	bDone									:BOOL;
	bBusy									:BOOL;
	bErr									:BOOL;
	nErrID									:UDINT;
	
END_VAR
VAR_IN_OUT

	stAxis									:Tc2_MC2.Axis_Ref;

END_VAR
VAR
	
	eStateRevSeq							:E_AxisReversingSequence;
	eRevSeqErrStep							:E_AxisReversingSequence := eAxisRevSeq_NoError;
	fbTimerIdleTime							:TON;
	fbMoveAbsolute							:Tc2_MC2.MC_MoveAbsolute;
	fbStop									:Tc2_MC2.MC_Stop;

END_VAR
(* End *)

(* Reversing sequence axis *)

	CASE eStateRevSeq OF

		eAxisRevSeq_Start			:	(* Wait for start *)
		
			bDone := FALSE;
			bBusy := FALSE;
			
			IF bStart
			THEN

				bBusy 		 := TRUE;
				eStateRevSeq := eAxisRevSeq_Init;
				
			END_IF		


		eAxisRevSeq_Init			:	(* Initialize *)
		
			fbMoveAbsolute(
				Axis	 := stAxis, 
				Execute	 := FALSE);
				
			fbTimerIdleTime(
				IN	 	 :=	FALSE);
			
			fbStop(
				Axis	 :=	stAxis,
				Execute	 :=	FALSE);
				
			eStateRevSeq := eAxisRevSeq_AxisStartPos1;


		eAxisRevSeq_AxisStartPos1	:	(* Start axis to position 1 *)
		
			fbMoveAbsolute(
				Axis		:= stAxis, 
				Execute		:= TRUE, 
				Position	:= fTargetPosition1, 
				Velocity	:= fTargetVelocity1, 
				ErrorID		=> nErrID);
			
		
			IF NOT fbMoveAbsolute.Busy
				AND NOT fbMoveAbsolute.Error
			THEN
			
				fbMoveAbsolute(
					Axis		:= stAxis, 
					Execute		:= FALSE);
				eStateRevSeq := eAxisRevSeq_IdleTime1;

			ELSIF bStop
			THEN

				fbMoveAbsolute(
					Axis	 := stAxis, 
					Execute	 := FALSE);
				eStateRevSeq := eAxisRevSeq_AxisStop;

			ELSIF NOT fbMoveAbsolute.Busy
					AND fbMoveAbsolute.Error
			THEN

				eRevSeqErrStep := eStateRevSeq;
				eStateRevSeq   := eAxisRevSeq_ErrorStep;

			END_IF


		eAxisRevSeq_IdleTime1		:	(* delayed restart *)
		
			fbTimerIdleTime(
				IN	:=	TRUE, 
				PT	:= 	tIdleTime);

			IF NOT bStop			
				AND fbTimerIdleTime.Q 
			THEN

				fbTimerIdleTime(IN	:=	FALSE);
				eStateRevSeq := eAxisRevSeq_AxisStartPos2;

			ELSIF bStop
			THEN

				eStateRevSeq := eAxisRevSeq_Done;

			END_IF


		eAxisRevSeq_AxisStartPos2	:	(* Start axis to position 2 *)
		
			fbMoveAbsolute(
				Axis		:= stAxis, 
				Execute		:= TRUE, 
				Position	:= fTargetPosition2, 
				Velocity	:= fTargetVelocity2, 
				ErrorID		=> nErrID);
			
		
			IF NOT fbMoveAbsolute.Busy
				AND NOT fbMoveAbsolute.Error
			THEN
				fbMoveAbsolute(
					Axis	 := stAxis, 
					Execute	 := FALSE);
				eStateRevSeq := eAxisRevSeq_IdleTime2;

			ELSIF bStop
			THEN

				fbMoveAbsolute(
					Axis		:= stAxis, 
					Execute	:= FALSE);
				eStateRevSeq := eAxisRevSeq_AxisStop;

			ELSIF NOT fbMoveAbsolute.Busy
					AND fbMoveAbsolute.Error
			THEN

				eRevSeqErrStep := eStateRevSeq;
				eStateRevSeq   := eAxisRevSeq_ErrorStep;

			END_IF		


		eAxisRevSeq_IdleTime2		:	(* delayed restart*)

			fbTimerIdleTime(
				IN	:=	TRUE, 
				PT	:= 	tIdleTime);
				
			IF NOT bStop			
				AND fbTimerIdleTime.Q 
			THEN

				fbTimerIdleTime(IN	:=	FALSE);
				eStateRevSeq := eAxisRevSeq_Done;
				
			ELSIF bStop
			THEN
			
				eStateRevSeq := eAxisRevSeq_Done;
				
			END_IF
			
			
		eAxisRevSeq_AxisStop		:	(* Stop axis *)

			fbStop(
				Axis	:=	stAxis, 
				Execute	:=	TRUE, 
				ErrorID	=>	nErrID );
				
			IF (fbStop.Done
				OR fbStop.CommandAborted)
				AND NOT fbStop.Error
			THEN
				fbStop(
					Axis	:=	stAxis, 
					Execute	:=	FALSE);
				eStateRevSeq := eAxisRevSeq_Done;

			ELSIF NOT fbStop.Busy
					AND fbStop.Error
			THEN

				eRevSeqErrStep := eStateRevSeq;
				eStateRevSeq   := eAxisRevSeq_ErrorStep;

			END_IF			
				
			
		eAxisRevSeq_Done			:	(* Sequence done *)

			bDone := TRUE;
			
			IF NOT bStart
				AND NOT bStop
			THEN
				bDone 		 := FALSE;
				bBusy 		 := FALSE;
				eStateRevSeq := eAxisRevSeq_Start;
				
			ELSIF bStart
				AND NOT bStop
			THEN
				bDone 		 := FALSE;
				eStateRevSeq := eAxisRevSeq_AxisStartPos1;
			END_IF

			
		eAxisRevSeq_ErrorStep		:	(* Error step *)
		
			bErr := TRUE;
			nErrID;
			
			IF NOT bStart
				AND NOT bStop
			THEN
				bErr 		   := FALSE;
				nErrID		   := 0;
				eRevSeqErrStep := eAxisRevSeq_NoError;
				eStateRevSeq   := eAxisRevSeq_Start;
			END_IF

	ELSE

		(* If not a valid step is active, then put on start *)
		eRevSeqErrStep := eAxisRevSeq_NoError;
		eStateRevSeq   := eAxisRevSeq_Start;

	END_CASE

(* End *)

END_FUNCTION_BLOCK

// ---- POUs/Motion/Axis2.TcPOU
PROGRAM Axis2
VAR
	
	sAxisDescription						:STRING	:= 'Axis 2 - EL7201 - AM8111-0F20';	

(* Axis - basic functions *)
	fbAxis									:FB_Axis;
	fMoveAbsPosition						:LREAL;				(* Target position *)
	fMoveAbsVelocity						:LREAL	:= 500.0;	(* Target speed axis 2 max. 10000.0 Degree/s *)
	bStartMoveAbs							:BOOL;
	bMoveAbsBusy							:BOOL;
	bMoveAbsDone							:BOOL;
	bAxisErr								:BOOL;
	nAxisErrId								:DWORD;
	bReset									:BOOL;
	bStop									:BOOL;
	bStopAxisDone							:BOOL;
	bStopAxisBusy							:BOOL;
	bRevSeqStart							:BOOL;
	bStartparameterSet						:BOOL;
	
(* Test - change target position - Axis *)
	bTestChangeTargetPos					:BOOL;				(* Test - change target position *)
	bMaxPositionReached						:BOOL;

(* Couple Axis on Handwheel) *)
	fbGearIn								:Tc2_MC2.MC_GearIn;
	bGearInDone								:BOOL;
	bAxisCoupled							:BOOL;

(* Uncouple Axis *)
	fbGearOut								:Tc2_MC2.MC_GearOut;
	bGearOutDone							:BOOL;

END_VAR
(* End *)

(* Axis 2 *)

(* Axis - basic functions  *)

	IF NOT bStartparameterSet
	THEN
		(* Startup Parameter reversing sequence *)
		fbAxis.fRevSeqTargetPos1	:= 1800.0;
		fbAxis.fRevSeqTargetVelo1	:= 1500.0;
		fbAxis.fRevSeqTargetPos2	:= 0.0;
		fbAxis.fRevSeqTargetVelo2	:= 200.0;
		fbAxis.nRevSeqIdleTime		:= 500;
		bStartparameterSet			:=TRUE;
	END_IF
		
	fbAxis(
		bPowerEnable		:= 	bSwitchS13,
		fPowerOverride		:= 	F_Scaling(nAnalogInR10, 100.0, 32767.0),
		bMoveAbsExecute		:= 	(bStartMoveAbs OR bSwitchS16) AND NOT stAxis2.Status.Coupled,
		fMoveAbsPosition	:= 	fMoveAbsPosition,
		fMoveAbsVelocity	:= 	fMoveAbsVelocity,
		bReset				:= 	bReset OR bSwitchS21,
		bStopAxis			:= 	bStop,
		bRevSeqStart		:=  (bSwitchS20 OR bRevSeqStart) AND fbAxis.bPowerStatus, 
		stAxis				:= 	stAxis2,
		bPowerStatus		=> 	bLedH13,
		bMoveAbsDone		=> 	bMoveAbsDone,
		bMoveAbsBusy		=> 	bMoveAbsBusy,
		bAxisErr			=> 	bAxisErr,
		nAxisErrId			=> 	nAxisErrId,
		bStopAxisDone		=> 	bStopAxisDone,
		bStopAxisBusy		=> 	bStopAxisBusy);

(* Test - change target position - Axis *)
	IF bTestChangeTargetPos
		AND (fMoveAbsPosition <= stAxis2.NcToPlc.ActPos)
			AND NOT bMaxPositionReached
	THEN
		fMoveAbsPosition := fMoveAbsPosition + 180.0;
	ELSE
		IF bTestChangeTargetPos
			AND (fMoveAbsPosition >= 3600.0)
		THEN
			fMoveAbsPosition 	:= 0.0;
			bMaxPositionReached	:= TRUE;
		END_IF
	END_IF

	IF bTestChangeTargetPos
		AND (stAxis2.NcToPlc.ActPos < 1.0)
	THEN
		bMaxPositionReached	:= FALSE;
	END_IF

	IF bSwitchS17
	THEN
		bMaxPositionReached	:= FALSE;
		fMoveAbsPosition 	:= 0.0;
	END_IF
	
(* Couple Axis on Handwheel *)
	fbGearIn(
		Execute			:= 	bHandwheelSwitchS28,
		RatioNumerator	:= 	1,
		RatioDenominator:= 	1,
		Acceleration	:= 	,
		Deceleration	:= 	,
		Jerk			:= 	,
		BufferMode		:= 	,
		Options			:= 	,
		Master			:= 	stAxis5,
		Slave			:= 	stAxis2,
		InGear			=> 	bGearInDone,
		Busy			=> 	,
		Active			=> 	,
		CommandAborted	=> 	,
		Error			=> 	,
		ErrorID			=> 	);

(* Axis coupled *)
	bAxisCoupled := stAxis2.Status.Coupled;

(* Uncouple Axis *)
	fbGearOut(
		Execute	:= 	bSwitchS17,
		Options	:= 	,
		Slave	:= 	stAxis2,
		Done	=> 	bGearOutDone,
		Busy	=> 	,
		Error	=> 	,
		ErrorID	=> 	);
	
(* End *)

END_PROGRAM

// ---- POUs/Motion/Axis3.TcPOU
PROGRAM Axis3
VAR
	
	sAxisDescription						:STRING	:= 'Axis 3 - AX5203-A - AM8111-0F10';	

(* Axis - basic functions *)
	fbAxis									:FB_AxisAX5xxx;
	fMoveAbsPosition						:LREAL;				(* Target position *)
	fMoveAbsVelocity						:LREAL	:= 500.0;	(* Target speed axis 3 max. 18000.0 Degree/s *)
	bStartMoveAbs							:BOOL;
	bMoveAbsBusy							:BOOL;
	bMoveAbsDone							:BOOL;
	bAxisErr								:BOOL;
	nAxisErrId								:DWORD;
	bReset									:BOOL;
	bStop									:BOOL;
	bStopAxisDone							:BOOL;
	bStopAxisBusy							:BOOL;
	bRevSeqStart							:BOOL;
	bStartparameterSet						:BOOL;
	
(* Test - change target position - Axis 3 *)
	bTestChangeTargetPos					:BOOL;				(* Test - change target position *)
	bMaxPositionReached						:BOOL;	

(* Couple Axis 3 on Axis 5 (Handwheel) *)
	fbGearIn								:Tc2_MC2.MC_GearIn;
	bGearInDone								:BOOL;
	bAxisCoupled							:BOOL;

(* Uncouple Axis 3 *)
	fbGearOut								:Tc2_MC2.MC_GearOut;
	bGearOutDone							:BOOL;
	
(*Superimposed and Buffered Moves*)
	mv_Axis3Abs : Tc2_MC2.MC_MoveAbsolute;
	mv_Axis3Rel : Tc2_MC2.MC_MoveRelative;
	iMstrMvMode2	: INT;
	bMvMstr2		: BOOL;
	lrMstrTarg2		: LREAL := 90;
	lrMstrVelo2		: LREAL := 10;
	mv_MasterSprImp	: Tc2_MC2.MC_MoveSuperImposed;
	bMvMstr3		: BOOL;
	lrMstrTarg3		: LREAL := 90;

END_VAR
(* End *)

(* Axis 3 *)

(* Axis - basic functions  *)

	IF NOT bStartparameterSet
	THEN
		(* Startup Parameter reversing sequence *)
		fbAxis.fRevSeqTargetPos1	:= 720.0;
		fbAxis.fRevSeqTargetVelo1	:= 5000.0;
		fbAxis.fRevSeqTargetPos2	:= 0.0;
		fbAxis.fRevSeqTargetVelo2	:= 5000.0;
		fbAxis.nRevSeqIdleTime		:= 250;
		bStartparameterSet			:=TRUE;
	END_IF
		
	fbAxis(
		bPowerEnable		:= 	bSwitchS14,
		fPowerOverride		:= 	F_Scaling(aOsAnalogInR11[0], 100.0, 32767.0),
		bMoveAbsExecute		:= 	(bStartMoveAbs OR bSwitchS16) AND NOT stAxis3.Status.Coupled,
		fMoveAbsPosition	:= 	fMoveAbsPosition,
		fMoveAbsVelocity	:= 	fMoveAbsVelocity,
		bReset				:= 	bReset OR bSwitchS21,
		bStopAxis			:= 	bStop,
		bRevSeqStart		:=  (bSwitchS20 OR bRevSeqStart) AND fbAxis.bPowerStatus, 
		stAxis				:= 	stAxis3,
		bPowerStatus		=> 	bLedH14,
		bMoveAbsDone		=> 	bMoveAbsDone,
		bMoveAbsBusy		=> 	bMoveAbsBusy,
		bAxisErr			=> 	bAxisErr,
		nAxisErrId			=> 	nAxisErrId,
		bStopAxisDone		=> 	bStopAxisDone,
		bStopAxisBusy		=> 	bStopAxisBusy);

(* Test - change target position - Axis *)
	IF bTestChangeTargetPos
		AND (fMoveAbsPosition <= stAxis3.NcToPlc.ActPos)
			AND NOT bMaxPositionReached
	THEN
		fMoveAbsPosition := fMoveAbsPosition + 180.0;
	ELSE
		IF bTestChangeTargetPos
			AND (fMoveAbsPosition >= 3600.0)
		THEN
			fMoveAbsPosition 	:= 0.0;
			bMaxPositionReached	:= TRUE;
		END_IF
	END_IF

	IF bTestChangeTargetPos
		AND (stAxis3.NcToPlc.ActPos < 1.0)
	THEN
		bMaxPositionReached	:= FALSE;
	END_IF

	IF bSwitchS17
	THEN
		bMaxPositionReached	:= FALSE;
		fMoveAbsPosition 	:= 0.0;
	END_IF
	
(* Couple Axis on Handwheel *)
	fbGearIn(
		Execute			:= 	bHandwheelSwitchS28,
		RatioNumerator	:= 	1,
		RatioDenominator:= 	1,
		Acceleration	:= 	,
		Deceleration	:= 	,
		Jerk			:= 	,
		BufferMode		:= 	,
		Options			:= 	,
		Master			:= 	stAxis5,
		Slave			:= 	stAxis3,
		InGear			=> 	bGearInDone,
		Busy			=> 	,
		Active			=> 	,
		CommandAborted	=> 	,
		Error			=> 	,
		ErrorID			=> 	);

(* Axis coupled *)
	bAxisCoupled := stAxis3.Status.Coupled;

(* Uncouple Axis *)
	fbGearOut(
		Execute	:= 	bSwitchS17,
		Options	:= 	,
		Slave	:= 	stAxis3,
		Done	=> 	bGearOutDone,
		Busy	=> 	,
		Error	=> 	,
		ErrorID	=> 	);

		
(*Buffered Move*)
	mv_Axis3Abs(
		Axis:= stAxis3, 
		Execute:= iMstrMvMode2=0 AND bMvMstr2, 
		Position:= lrMstrTarg2, 
		Velocity:= lrMstrVelo2);
		
	mv_Axis3Rel(	
		Axis:= stAxis3, 
		Execute:= iMstrMvMode2=1 AND bMvMstr2, 
		Distance:= lrMstrTarg2, 
		Velocity:= lrMstrVelo2);
		
IF (NOT(mv_Axis3Abs.Busy) AND NOT(mv_Axis3Rel.busy)) THEN
	bMvMstr2:=FALSE;
END_IF

(*Superimposed Move*)
mv_MasterSprImp(
	Axis:= stAxis3, 
	Execute:= bMvMstr3, 
	Mode:= SUPERPOSITIONMODE_VELOREDUCTION_ADDITIVEMOTION, 
	Distance:= lrMstrTarg3, 
	// assume max velo is 2000 (config parameter)
	VelocityDiff:= 2000-stAxis3.NcToPlc.SetVelo, 
	Acceleration:= , 
	Deceleration:= , 
	Jerk:= , 
	VelocityProcess:= stAxis3.NcToPlc.SetVelo, 
	// use 75% of remaining distance to 'catch up'
	Length:= (stAxis3.NcToPlc.TargetPos-stAxis3.NcToPlc.ActPos)*0.75);
			
(* End *)

END_PROGRAM

// ---- POUs/Motion/Components/FB_AxisAX5xxx.TcPOU
FUNCTION_BLOCK FB_AxisAX5xxx
VAR_INPUT

	bPowerEnable							:BOOL;
	fPowerOverride							:LREAL;
	bMoveAbsExecute							:BOOL;
	fMoveAbsPosition						:LREAL;
	fMoveAbsVelocity						:LREAL;
	bReset									:BOOL;
	bStopAxis								:BOOL;
	bRevSeqStart							:BOOL;
	bRevSeqStop								:BOOL;
	fRevSeqTargetPos1						:LREAL; 
	fRevSeqTargetVelo1						:LREAL;	 
	fRevSeqTargetPos2						:LREAL;	 
	fRevSeqTargetVelo2						:LREAL; 
	nRevSeqIdleTime							:UINT;
	
END_VAR
VAR_OUTPUT

	bPowerStatus							:BOOL;
	bMoveAbsDone							:BOOL;
	bMoveAbsBusy							:BOOL;
	bAxisErr								:BOOL;
	nAxisErrId								:DWORD;
	bStopAxisDone							:BOOL;
	bStopAxisBusy							:BOOL;
	bRevSeqDone								:BOOL;
	bRevSeqBusy								:BOOL;
	
END_VAR
VAR_IN_OUT

	stAxis									:Tc2_Mc2.Axis_Ref;

END_VAR
VAR

	fbMcPower								:Tc2_MC2.MC_Power;
	fbMoveAbsolute							:Tc2_MC2.MC_MoveAbsolute;
	fbReadAxisError							:Tc2_MC2.MC_ReadAxisError;
	fbReset									:MC_Reset_Ax5xxx;
	fbStop									:Tc2_MC2.MC_Stop;
	fbReversingSequence						:FB_ReversingSequence;

END_VAR
(* End *)

(* FB_Axis AX5xxx *)

(* Read status of the axis *)
	stAxis.ReadStatus();

(* Enable axis *)
	fbMcPower(
		Enable			:= 	bPowerEnable,
		Enable_Positive	:= 	bPowerEnable,
		Enable_Negative	:= 	bPowerEnable,
		Override		:= 	fPowerOverride,
		Axis			:= 	stAxis,
		Status			=> 	bPowerStatus);

(* Start axis at an absolute position *)
	fbMoveAbsolute(
		Execute		:=	bMoveAbsExecute,
		Position	:=	fMoveAbsPosition,
		Velocity	:=	fMoveAbsVelocity,
		Axis		:=	stAxis,
		Done		=>	bMoveAbsDone,
		Busy		=>	bMoveAbsBusy);

(* Read the error code of the axis *)
	fbReadAxisError(
		Enable		:=	TRUE,
		Axis		:=	stAxis,
		AxisErrorID	=>	nAxisErrId);

	bAxisErr := nAxisErrId <> 0;

(* Reset axis in case of failure *)
	fbReset(
		Execute		:= 	bReset,
		Axis		:= 	stAxis);

(* Stop axis *)
	fbStop(
		Execute 	:=	bStopAxis,
		Axis		:=	stAxis,
		Done		=>	bStopAxisDone,
		Busy		=>	bStopAxisBusy);

(* Axis reversing sequence *)	
	fbReversingSequence(
		bStart				:= 	bRevSeqStart,
		bStop				:= 	bRevSeqStop,
		fTargetPosition1	:= 	fRevSeqTargetPos1,
		fTargetVelocity1	:= 	fRevSeqTargetVelo1,
		fTargetPosition2	:= 	fRevSeqTargetPos2,
		fTargetVelocity2	:= 	fRevSeqTargetVelo2,
		tIdleTime			:= 	TO_TIME(nRevSeqIdleTime),
		bDone				=> 	bRevSeqDone,
		bBusy				=> 	bRevSeqBusy,
		bErr				=> 	,
		nErrID				=> 	,
		stAxis				:= 	stAxis);
		
(* End *)

END_FUNCTION_BLOCK

// ---- POUs/Motion/Components/MC_Reset_Ax5xxx.TcPOU
FUNCTION_BLOCK MC_Reset_Ax5xxx
VAR_INPUT

	Execute									:BOOL;

END_VAR
VAR_IN_OUT

	Axis	 								:Tc2_Mc2.AXIS_REF;

END_VAR
VAR_OUTPUT

	Done									:BOOL;
	Busy									:BOOL;
	Error									:BOOL;
	ErrorId									:DWORD;

END_VAR
VAR

	bDriveProtected							:BOOL;
	bDriveDeviceError						:BOOL;
	bDriveIoDataInvalid						:BOOL;
	bDriveError								:BOOL;

	fbNcReset								:Tc2_Mc2.MC_Reset;
	fbSoEReset								:FB_SoEReset;

	eStateResetSeq							:E_McResetStatus;
	eResetSeqErrStep						:E_McResetStatus := eMcReset_NoError;

END_VAR
(* End *)

(* MC_Reset_Ax5xxx *)

(* Evaluate messages *)
	bDriveProtected 	:= TO_BOOL(Axis.NcToPlc.StateDWord.5);
	bDriveDeviceError   := TO_BOOL(Axis.NcToPlc.StateDWord.28);
	bDriveIoDataInvalid	:= TO_BOOL(Axis.NcToPlc.StateDWord.30);
	bDriveError			:= TO_BOOL(Axis.NcToPlc.StateDWord.31);

	
(* Reset sequence *)
	CASE eStateResetSeq OF
	
		eMcReset_Start			:	(* Wait for start *)
		
				Busy := FALSE;
				Done := FALSE;
	
				IF Execute
				THEN
				
					Busy := TRUE;
					eStateResetSeq := eMcReset_Init;

				END_IF


		eMcReset_Init			:	(* Initialize *)
			
				fbSoEReset(	
					NetId		:=	'',
					Execute		:=	FALSE,
					Timeout		:=	T#12S,
					Axis		:=	Axis);

				fbNcReset(	
					Execute		:=	FALSE,
					Axis		:=	Axis);

				eStateResetSeq 		:= eMcReset_ResetHardware;

	
		eMcReset_ResetHardware	:	(* Reset hardware *)
		
				fbSoEReset(	
					NetId	:=	'' ,
					Execute	:=	Execute
									AND (bDriveDeviceError
										OR bDriveIoDataInvalid),
					Timeout	:=	T#12S ,
					Axis	:=	Axis);
	
				IF NOT fbSoEReset.Busy
					AND NOT fbSoEReset.Error
				THEN
	
					fbSoEReset(	
						NetId	:=	'',
						Execute	:=	FALSE,
						Timeout	:=	T#12S,
						Axis	:=	Axis);
	
					eStateResetSeq := eMcReset_ResetNc;
	
				ELSIF NOT fbSoEReset.Busy
					AND fbSoEReset.Error
				THEN

					eResetSeqErrStep := eStateResetSeq;
					eStateResetSeq   := eMcReset_ErrorStep;
	
				END_IF


		eMcReset_ResetNc		:	(* Reset NC *)
		
				fbNcReset(	
					Execute	:=	Execute
									AND bDriveError
										AND NOT bDriveDeviceError
											AND NOT fbSoEReset.Busy
												AND NOT bDriveProtected,
					Axis	:=	Axis);
	
				IF NOT fbNcReset.Busy
					AND NOT fbNcReset.Error
				THEN
	
					fbNcReset(	
						Execute	:=	FALSE,
						Axis	:=	Axis);
	
					eStateResetSeq := eMcReset_Done;

				ELSIF NOT fbNcReset.Busy
					AND fbNcReset.Error
				THEN

					eResetSeqErrStep := eStateResetSeq;
					eStateResetSeq   := eMcReset_ErrorStep;
	
				END_IF
				
	
		eMcReset_Done			:	(* Reset done *)
		
				Busy := FALSE;
				Done := TRUE;
	
				IF NOT Execute
				THEN
					eStateResetSeq := eMcReset_Start;
				END_IF


		eMcReset_ErrorStep			:	(* Error step *)

			IF NOT Execute
			THEN
				eResetSeqErrStep := eMcReset_NoError;
				eStateResetSeq   := eMcReset_Start;
			END_IF


	ELSE

		(* If not a valid step is active, then put on start *)
		eResetSeqErrStep := eMcReset_NoError;
		eStateResetSeq 	 := eMcReset_Start;

	END_CASE

	Error	:= bDriveError
					OR bDriveDeviceError;

	ErrorId	:= Axis.NcToPlc.ErrorCode;

(* End *)

END_FUNCTION_BLOCK

// ---- POUs/Motion/Axis4.TcPOU
PROGRAM Axis4
VAR
	
	sAxisDescription						:STRING	:= 'Axis 4 - AX5203-B - AM8111-0F21';	

(* Axis - basic functions *)
	fbAxis									:FB_AxisAX5xxx;
	fMoveAbsPosition						:LREAL;				(* Target position *)
	fMoveAbsVelocity						:LREAL	:= 500.0;	(* Target speed axis 3 max. 18000.0 Degree/s *)
	bStartMoveAbs							:BOOL;
	bMoveAbsBusy							:BOOL;
	bMoveAbsDone							:BOOL;
	bAxisErr								:BOOL;
	nAxisErrId								:DWORD;
	bReset									:BOOL;
	bStop									:BOOL;
	bStopAxisDone							:BOOL;
	bStopAxisBusy							:BOOL;
	bRevSeqStart							:BOOL;
	bStartparameterSet						:BOOL;
	
(* Test - change target position - Axis 4 *)
	bTestChangeTargetPos					:BOOL;				(* Test - change target position *)
	bMaxPositionReached						:BOOL;
		
(* Couple Axis 4 on Axis 5 (Handwheel) *)
	fbGearIn								:Tc2_MC2.MC_GearIn;
	bGearInDone								:BOOL;
	bAxisCoupled							:BOOL;

(* Uncouple Axis 4 *)
	fbGearOut								:Tc2_MC2.MC_GearOut;
	bGearOutDone							:BOOL;
	
END_VAR
(* End *)

(* Axis 4 *)

(* Axis - basic functions  *)	

	IF NOT bStartparameterSet
	THEN
		(* Startup Parameter reversing sequence *)
		fbAxis.fRevSeqTargetPos1	:= 7200.0;
		fbAxis.fRevSeqTargetVelo1	:= 9000.0;
		fbAxis.fRevSeqTargetPos2	:= 0.0;
		fbAxis.fRevSeqTargetVelo2	:= 5000.0;
		fbAxis.nRevSeqIdleTime		:= 600;
		bStartparameterSet			:=TRUE;
	END_IF
		
	fbAxis(
		bPowerEnable		:= 	bSwitchS15,
		fPowerOverride		:= 	F_Scaling(aOsAnalogInR11[0], 100.0, 32767.0),
		bMoveAbsExecute		:= 	(bStartMoveAbs OR bSwitchS16) AND NOT stAxis4.Status.Coupled,
		fMoveAbsPosition	:= 	fMoveAbsPosition,
		fMoveAbsVelocity	:= 	fMoveAbsVelocity,
		bReset				:= 	bReset OR bSwitchS21,
		bStopAxis			:= 	bStop,
		bRevSeqStart		:=  (bSwitchS20 OR bRevSeqStart) AND fbAxis.bPowerStatus, 
		stAxis				:= 	stAxis4,
		bPowerStatus		=> 	bLedH15,
		bMoveAbsDone		=> 	bMoveAbsDone,
		bMoveAbsBusy		=> 	bMoveAbsBusy,
		bAxisErr			=> 	bAxisErr,
		nAxisErrId			=> 	nAxisErrId,
		bStopAxisDone		=> 	bStopAxisDone,
		bStopAxisBusy		=> 	bStopAxisBusy);

(* Test - change target position - Axis *)
	IF bTestChangeTargetPos
		AND (fMoveAbsPosition <= stAxis4.NcToPlc.ActPos)
			AND NOT bMaxPositionReached
	THEN
		fMoveAbsPosition := fMoveAbsPosition + 180.0;
	ELSE
		IF bTestChangeTargetPos
			AND (fMoveAbsPosition >= 3600.0)
		THEN
			fMoveAbsPosition 	:= 0.0;
			bMaxPositionReached	:= TRUE;
		END_IF
	END_IF

	IF bTestChangeTargetPos
		AND (stAxis4.NcToPlc.ActPos < 1.0)
	THEN
		bMaxPositionReached	:= FALSE;
	END_IF

	IF bSwitchS17
	THEN
		bMaxPositionReached	:= FALSE;
		fMoveAbsPosition	:= 0.0;
	END_IF
	
(* Couple Axis on Handwheel *)
	fbGearIn(
		Execute			:= 	bHandwheelSwitchS28,
		RatioNumerator	:= 	1,
		RatioDenominator:= 	1,
		Acceleration	:= 	,
		Deceleration	:= 	,
		Jerk			:= 	,
		BufferMode		:= 	,
		Options			:= 	,
		Master			:= 	stAxis5,
		Slave			:= 	stAxis4,
		InGear			=> 	bGearInDone,
		Busy			=> 	,
		Active			=> 	,
		CommandAborted	=> 	,
		Error			=> 	,
		ErrorID			=> 	);

(* Axis coupled *)
	bAxisCoupled := stAxis4.Status.Coupled;

(* Uncouple Axis *)
	fbGearOut(
		Execute	:= 	bSwitchS17,
		Options	:= 	,
		Slave	:= 	stAxis4,
		Done	=> 	bGearOutDone,
		Busy	=> 	,
		Error	=> 	,
		ErrorID	=> 	);
			
(* End *)

END_PROGRAM

// ---- POUs/MC3/ReversingSequence/MC3_ReversingSequence.TcPOU
PROGRAM MC3_ReversingSequence
VAR
	bStart:		BOOL;
	ax1:		Tc3_Mc3Ptp.AXIS_REF;
	fbPower:	Tc3_Mc3Ptp.MC_Power;		
	fbMoveAbs:	Tc3_Mc3Ptp.MC_MoveAbsolute;	
	timer:		TON;
	nState:		INT :=0;
END_VAR

fbPower
(
	Axis:=ax1,
	Enable:=,
	EnableNegative:=TRUE,
	EnablePositive:=TRUE,
);
	

CASE nState OF
	0:
	IF bStart THEN
		fbPower.Enable:=TRUE;
		nState:=nState+1;
	END_IF

	1:
	IF fbPower.Status THEN
		fbMoveAbs.Position:=4000.0;
		fbMoveAbs.Velocity:=1000.0;
		fbMoveAbs.Execute:=TRUE;
		nState:=nState+1;
	END_IF
	
	2:
	IF NOT fbMoveAbs.Busy THEN
		IF fbMoveAbs.Done THEN
			fbMoveAbs.Execute:=FALSE;
			timer.PT:=T#1S;
			timer.IN:=TRUE;
			nState:=nState+1;
		END_IF
	END_IF
	
	3:
	IF timer.Q THEN
		timer.IN:=FALSE;
		fbMoveAbs.Position:=0000.0;
		fbMoveAbs.Velocity:=1000.0;
		fbMoveAbs.Execute:=TRUE;
		nState:=nState+1;
	END_IF
	
	4:
	IF NOT fbMoveAbs.Busy THEN
		IF fbMoveAbs.Done THEN
			fbMoveAbs.Execute:=FALSE;
			timer.PT:=T#1S;
			timer.IN:=TRUE;
		nState:=nState+1;
		END_IF
	END_IF

	5:
	IF timer.Q THEN
		timer.IN:=FALSE;
		nState:=0;
	END_IF
	
END_CASE


fbMoveAbs(Axis:=ax1);
timer();

END_PROGRAM

// ---- POUs/MC3/ExternalSetpoint_Mc3_Nc2/ExtSetpoint_MC3_NC2.TcPOU
// External Setpoint Generation: MC3 slave following NC2 master
// An MC3 slave axis follows an NC2 master axis via a custom external setpoint generator
// (FB_ExtSg_FollowNcAxis) that reads the NC2 master setpoints each cycle.
// The axes are powered and the generator is activated on program start.
PROGRAM ExtSetpoint_MC3_NC2
VAR
		////NC Master
	fbPowerMaster	   : TC2_MC2.MC_Power;


	////MC3 Slave
	Mc3SlaveAxis	   : TC3_Mc3Ptp.AXIS_REF;
	fbPowerMC3Slave	   : Tc3_Mc3Ptp.MC_Power;
	fbActivateMc3ExtSg : Tc3_Mc3Ptp.MC_ActivateExternalSetpointGeneration;
	fbMc3FollowNc	   : FB_ExtSg_FollowNcAxis('ExtSg_FollowNcAxis');
END_VAR

// Master Axis
fbPowerMaster(Axis			  := Nc2MasterAxis,
			  Enable		  := TRUE,
			  Enable_Positive := TRUE,
			  Enable_Negative := TRUE);


//MC3 Slave Axis
fbPowerMC3Slave(Axis		   := Mc3SlaveAxis,
				Enable		   := TRUE,
				EnableNegative := TRUE,
				EnablePositive := TRUE);

fbActivateMc3ExtSg(Axis						 := Mc3SlaveAxis,
				   ExternalSetpointGenerator := fbMc3FollowNc,
				   AllowOtherContext		 := TRUE,
				   EnableDynamicChecks		 := FALSE);

END_PROGRAM

// ---- POUs/MC3/ExternalSetpoint_Mc3_Nc2/FB_ExtSg_FollowNcAxis.TcPOU
{attribute 'c++_compatible'}
FUNCTION_BLOCK FB_ExtSg_FollowNcAxis EXTENDS MC_ExternalSetpointGenerator IMPLEMENTS ITcMcExternalSetpointGenerator

{attribute 'TcTypeSystem'}
METHOD FB_init : BOOL
VAR_INPUT
	(*  if TRUE, the retain variables are initialized (warm start / cold start) *)
	bInitRetains	: BOOL;
	(*  if TRUE, the instance afterwards gets moved into the copy code (online change) *)
	bInCopyCode	: BOOL;
	sObjectName	: STRING;
END_VAR
END_METHOD

{attribute 'TcTypeSystem'}
METHOD FB_reinit : BOOL
SUPER^.FB_reinit();
END_METHOD

{attribute 'TcTypeSystem'}
{attribute 'c++_compatible'}
METHOD OnCyclicSetpointGeneration : HRESULT
VAR_INPUT
	invokeId		 : XWORD;
	timeInGeneration : LREAL;
	position		 : REFERENCE TO LREAL;
	velocity		 : REFERENCE TO LREAL;
	acceleration	 : REFERENCE TO LREAL;
END_VAR
//GenerateSetpoint implementation 
position				   := Nc2MasterAxis.NcToPlc.SetPos;
velocity				   := Nc2MasterAxis.NcToPlc.SetVelo;
acceleration			   := Nc2MasterAxis.NcToPlc.SetAcc;
OnCyclicSetpointGeneration := S_OK;
END_METHOD

END_FUNCTION_BLOCK

// ---- POUs/MC3/Gearing/MC3_Gearing.TcPOU
// Gearing sample
// Shows electronic gearing with MC_GearIn (stationary and velocity (master) coupling) and MC_GearInPos
// (position-synchronized coupling), plus error propagation between coupled axes.
// Operation: set 'Command' (E_Command) to Enable, then a GearIn* command
PROGRAM MC3_Gearing
VAR
	//
	Axis : ARRAY[0..(AXES_COUNT - 1)] OF Tc3_Mc3Ptp.AXIS_REF;

	//
	McPower		   : ARRAY[0..(AXES_COUNT - 1)] OF Tc3_Mc3Ptp.MC_Power;
	McReset		   : ARRAY[0..(AXES_COUNT - 1)] OF Tc3_Mc3Ptp.MC_Reset;
	McHalt		   : ARRAY[0..(AXES_COUNT - 1)] OF Tc3_Mc3Ptp. MC_Halt;
	McSetPosition  : ARRAY[0..(AXES_COUNT - 1)] OF Tc3_Mc3Ptp.MC_SetPosition;
	McMoveAbsolute : ARRAY[0..(AXES_COUNT - 1)] OF Tc3_Mc3Ptp.MC_MoveAbsolute;
	McMoveVelocity : ARRAY[0..(AXES_COUNT - 1)] OF Tc3_Mc3Ptp.MC_MoveVelocity;

	//
	McGearIn					: Tc3_Mc3Ptp.MC_GearIn;
	McGearInPos					: Tc3_Mc3Ptp.MC_GearInPos;
	WaitForStableActualPosition : Tc3_Mc3Ptp.MC_WaitForStableActualPosition;

	//
	i		 : UDINT;
	Sequence : UDINT;
	Command	 : E_GearCommand;
	ErrorId	 : UDINT;

	// Error Testing
	TriggerMasterError	  : BOOL;
	TriggerSlaveError	  : BOOL;
	ControlError		  : BOOL				   := TRUE;
	ReactionToMasterError : EReactionToMasterError := EReactionToMasterError.TriggerSlaveError;
	ReactionToSlaveError  : EReactionToSlaveError  := EReactionToSlaveError.TriggerMasterError;
	McTriggerMasterError  : Tc3_Mc3Ptp.MC_TriggerError;
	McTriggerSlaveError	  :Tc3_Mc3Ptp. MC_TriggerError;
END_VAR

VAR CONSTANT
	AXES_COUNT : UDINT := 2;
END_VAR

(* Commands:
    1- Enable
       2 - GearInStationary ( MC_GearIn )
	   3 - GearInVelocity   ( MC_GearIn )
	   4 - GearInPosition   ( MC_GearInPos )
    5 - Disable 
*)
CASE Sequence OF
	0:
		IF Command = E_GearCommand.Enable THEN
			NextStep(Sequence);
		END_IF

	10:
		IF Enable() THEN
			Command := E_GearCommand.Idle;
			SetStep(Sequence, 100);
		END_IF

	100:
		IF Command = E_GearCommand.Disable THEN
			SetStep(Sequence, 1000);
		END_IF

		IF Command = E_GearCommand.GearInStationary THEN
			SetStep(Sequence, 200);
		END_IF

		IF Command = E_GearCommand.GearInVelocity THEN
			SetStep(Sequence, 300);
		END_IF

		IF Command = E_GearCommand.GearInPosition THEN
			SetStep(Sequence, 400);
		END_IF

	200:
		IF GearInStationary() THEN
			SetStep(Sequence, 500);
		END_IF

	300:
		IF GearInVelocity() THEN
			SetStep(Sequence, 500);
		END_IF

	400:
		IF GearInPosition() THEN
			SetStep(Sequence, 500);
		END_IF

	500:
		IF Home() THEN
			Command := E_GearCommand.Idle;
			SetStep(Sequence, 100);
		END_IF

	1000:
		IF Disable() THEN
			Command := E_GearCommand.Idle;
			SetStep(Sequence, 0);
		END_IF
END_CASE

McTriggerMasterError(MotionObject := Axis[Master],
				 Execute	  := TriggerMasterError,
				 ErrorCode	  := 16#FFFFFFFF,
				 ControlError := ControlError,
				 Done		  =>,
				 Busy		  =>,
				 Error		  =>,
				 ErrorId	  =>);

McTriggerSlaveError(MotionObject := Axis[Slave],
				Execute		 := TriggerSlaveError,
				ErrorCode	 := 16#FFFFFFFF,
				ControlError := ControlError,
				Done		 =>,
				Busy		 =>,
				Error		 =>,
				ErrorId		 =>);

TriggerMasterError := TriggerSlaveError := FALSE;

METHOD Disable : BOOL
VAR_INPUT
END_VAR
McPower[Master](Axis		   := Axis[Master],
				Enable		   := FALSE,
				EnablePositive := FALSE,
				EnableNegative := FALSE,
				Status		   =>,
				Error		   =>,
				ErrorId		   =>);

McPower[Slave](Axis			  := Axis[Slave],
			   Enable		  := FALSE,
			   EnablePositive := FALSE,
			   EnableNegative := FALSE,
			   Status		  =>,
			   Error		  =>,
			   ErrorId		  =>);

Disable := NOT McPower[Master].Status AND NOT McPower[Slave].Status AND Axis[Master].McToPlc.Std.AxisState = EAxisState.Disabled AND Axis[Slave].McToPlc.Std.AxisState = EAxisState.Disabled;
END_METHOD

METHOD Enable : BOOL
VAR_INPUT
END_VAR
McPower[Master](Axis		   := Axis[Master],
				Enable		   := TRUE,
				EnablePositive := TRUE,
				EnableNegative := TRUE,
				Status		   =>,
				Error		   =>,
				ErrorId		   =>);

McPower[Slave](Axis			  := Axis[Slave],
			   Enable		  := TRUE,
			   EnablePositive := TRUE,
			   EnableNegative := TRUE,
			   Status		  =>,
			   Error		  =>,
			   ErrorId		  =>);

Enable := McPower[Master].Status AND McPower[Slave].Status AND Axis[Master].McToPlc.Std.AxisState = EAxisState.Standstill AND Axis[Slave].McToPlc.Std.AxisState = EAxisState.Standstill;
END_METHOD

METHOD GearInPosition : BOOL
VAR_INST
    GearInSequence : UDINT;
    //FB_
END_VAR
CASE GearInSequence OF
	0:
		McMoveAbsolute[Master].Position := 1000;
		McMoveAbsolute[Master].Execute	:= TRUE;
		IF McMoveAbsolute[Master].Busy THEN
			McMoveAbsolute[Master].Execute := FALSE;
			NextStep(GearInSequence);
		END_IF

	10: // Wait for Master to cover some distance as MC_GearInPos is instant in this version of MC3
		IF Axis[Master].McToPlc.Act.Position >= 250 THEN
			NextStep(GearInSequence);
		END_IF

	20:
		McGearInPos.Execute := TRUE;
		IF McGearInPos.InSync THEN
			McGearInPos.Execute := FALSE;
			NextStep(GearInSequence);
		END_IF

	30:
		WaitForStableActualPosition.Execute := TRUE;
		IF WaitForStableActualPosition.InPositionWindow AND WaitForStableActualPosition.Done AND NOT McMoveAbsolute[Master].Busy THEN
			McMoveAbsolute[Master].Execute		:= FALSE;
			WaitForStableActualPosition.Execute := FALSE;
			NextStep(GearInSequence);
		END_IF

	40:
		McHalt[Slave](Axis := Axis[Slave], Execute := TRUE);
		IF NOT McHalt[Slave].Busy AND McHalt[Slave].Done THEN
			McHalt[Slave](Axis := Axis[Slave], Execute := FALSE);
			NextStep(GearInSequence);
		END_IF

	50:
		SetStep(GearInSequence, 0);
		GearInPosition := TRUE;
END_CASE

McMoveAbsolute[Master](Axis			:= Axis[Master],
					   Velocity		:= 100,
					   Acceleration := 1000,
					   Deceleration := 500,
					   Jerk			:= 1000,
					   BufferMode	:= EBufferMode.Aborting);

McGearInPos(Master				  := Axis[Master],
			Slave				  := Axis[Slave],
			RatioNumerator		  := 1,
			RatioDenominator	  := 1,
			MasterSyncPosition	  := 500,
			SlaveSyncPosition	  := 250,
			Velocity			  := 1000,
			Acceleration		  := 1000,
			Deceleration		  := 1000,
			Jerk				  := 10000,
			BufferMode			  := EBufferMode.Aborting,
			ReactionToMasterError := ReactionToMasterError,
			ReactionToSlaveError  := ReactionToSlaveError,
			InSync				  =>,
			Busy				  =>,
			Active				  =>,
			CommandAborted		  =>,
			Error				  =>,
			ErrorId				  =>,
			MasterHasError		  =>);

WaitForStableActualPosition(Axis			  := Axis[Master],
							PositionTolerance := 0.001,
							WaitDuration	  := 0.5,
							TimeoutDuration	  := STRING_TO_LREAL('#Ignore'),
							InPositionWindow  =>,
							Done			  =>,
							Busy			  =>,
							Active			  =>,
							CommandAborted	  =>,
							Error			  =>,
							ErrorId			  =>);
END_METHOD

METHOD GearInStationary : BOOL
VAR_INST
    GearInSequence : UDINT;
END_VAR
CASE GearInSequence OF
	0:
		McGearIn.Execute := TRUE;
		IF McGearIn.InGear THEN
			McGearIn.Execute := FALSE;
			NextStep(GearInSequence);
		END_IF

	10:
		McMoveAbsolute[Master].Position := 1000;
		McMoveAbsolute[Master].Execute	:= TRUE;
		IF NOT McMoveAbsolute[Master].Busy AND McMoveAbsolute[Master].Done THEN
			McMoveAbsolute[Master].Execute := FALSE;
			NextStep(GearInSequence);
		END_IF

	20:
		McHalt[Slave](Axis := Axis[Slave], Execute := TRUE);
		IF NOT McHalt[Slave].Busy AND McHalt[Slave].Done THEN
			McHalt[Slave](Axis := Axis[Slave], Execute := FALSE);
			NextStep(GearInSequence);
		END_IF

	30:
		SetStep(GearInSequence, 0);
		GearInStationary := TRUE;
END_CASE

McGearIn(Master				   := Axis[Master],
		 Slave				   := Axis[Slave],
		 RatioNumerator		   := 1,
		 RatioDenominator	   := 2,
		 ReactionToMasterError := ReactionToMasterError,
		 ReactionToSlaveError  := ReactionToSlaveError);

McMoveAbsolute[Master](Axis			:= Axis[Master],
					   Velocity		:= 100,
					   Acceleration := 1000,
					   Deceleration := 500,
					   Jerk			:= 1000,
					   BufferMode	:= EBufferMode.Aborting);
END_METHOD

METHOD GearInVelocity : BOOL
VAR_INST
	GearInSequence : UDINT;
	WaitToGear	   : TON;
END_VAR
CASE GearInSequence OF
	0:
		McMoveVelocity[Master].Velocity := 100;
		McMoveVelocity[Master].Execute	:= TRUE;
		IF McMoveVelocity[Master].Busy AND McMoveVelocity[Master].InVelocity THEN
			McMoveVelocity[Master].Execute := FALSE;
			NextStep(GearInSequence);
		END_IF

	10:
		WaitToGear(IN := TRUE, PT := T#1S);
		IF WaitToGear.Q THEN
			WaitToGear(IN := FALSE);
			NextStep(GearInSequence);
		END_IF

	20:
		McGearIn.Execute := TRUE;
		IF McGearIn.InGear THEN
			McGearIn(Master := Axis[Master], Slave := Axis[Slave], Execute := FALSE);
			NextStep(GearInSequence);
		END_IF

	30:
		WaitToGear(IN := TRUE, PT := T#2S);
		IF WaitToGear.Q THEN
			WaitToGear(IN := FALSE);
			NextStep(GearInSequence);
		END_IF

	40:
		McMoveVelocity[Master](Axis			:= Axis[Master],
							   Execute		:= TRUE,
							   Velocity		:= 500,
							   Acceleration := 1000,
							   Deceleration := 1000,
							   Jerk			:= 10000,
							   BufferMode	:= EBufferMode.Aborting);

		IF McMoveVelocity[Master].Busy AND McMoveVelocity[Master].InVelocity THEN
			McMoveVelocity[Master](Axis := Axis[Master], Execute := FALSE);
			NextStep(GearInSequence);
		END_IF

	50:
		WaitToGear(IN := TRUE, PT := T#2S);
		IF WaitToGear.Q THEN
			WaitToGear(IN := FALSE);
			NextStep(GearInSequence);
		END_IF

	60:
		McMoveVelocity[Master](Axis			:= Axis[Master],
							   Execute		:= TRUE,
							   Velocity		:= 150,
							   Acceleration := 1000,
							   Deceleration := 1000,
							   Jerk			:= 10000,
							   BufferMode	:= EBufferMode.Aborting);

		IF McMoveVelocity[Master].Busy AND McMoveVelocity[Master].InVelocity THEN
			McMoveVelocity[Master](Axis := Axis[Master], Execute := FALSE);
			NextStep(GearInSequence);
		END_IF

	70:
		WaitToGear(IN := TRUE, PT := T#2S);
		IF WaitToGear.Q THEN
			WaitToGear(IN := FALSE);
			NextStep(GearInSequence);
		END_IF

	80:
		McHalt[Master](Axis := Axis[Master], Execute := TRUE);
		IF NOT McHalt[Master].Busy AND McHalt[Master].Done THEN
			McHalt[Master](Axis := Axis[Master], Execute := FALSE);
			NextStep(GearInSequence);
		END_IF

	90:
		McHalt[Slave](Axis := Axis[Slave], Execute := TRUE);
		IF NOT McHalt[Slave].Busy AND McHalt[Slave].Done THEN
			McHalt[Slave](Axis := Axis[Slave], Execute := FALSE);
			NextStep(GearInSequence);
		END_IF

	100:
		GearInSequence := 0;
		GearInVelocity := TRUE;
END_CASE

McGearIn(Master				   := Axis[Master],
		 Slave				   := Axis[Slave],
		 RatioNumerator		   := 1,
		 RatioDenominator	   := 2,
		 Acceleration		   := 1000,
		 Deceleration		   := 1000,
		 Jerk				   := 10000,
		 BufferMode			   := EBufferMode.Aborting,
		 ReactionToMasterError := ReactionToMasterError,
		 ReactionToSlaveError  := ReactionToSlaveError);

McMoveVelocity[Master](Axis			:= Axis[Master],
					   Acceleration := 1000,
					   Deceleration := 1000,
					   Jerk			:= 10000,
					   BufferMode	:= EBufferMode.Aborting);
END_METHOD

METHOD Home : BOOL
VAR_INST
    HomeSequence : UDINT;
END_VAR
CASE HomeSequence OF
	0:
		McSetPosition[Master](Axis	   := Axis[Master],
							  Execute  := TRUE,
							  Position := 0,
							  Relative := FALSE);

		IF McSetPosition[Master].Done AND NOT McSetPosition[Master].Busy THEN
			NextStep(HomeSequence);
		END_IF

	10:
		McSetPosition[Slave](Axis	  := Axis[Slave],
							 Execute  := TRUE,
							 Position := 0,
							 Relative := FALSE);

		IF McSetPosition[Slave].Done AND NOT McSetPosition[Slave].Busy THEN
			NextStep(HomeSequence);
		END_IF

	20:
		McSetPosition[Master](Axis := Axis[Master], Execute := FALSE, Position := 0);
		McSetPosition[Slave](Axis := Axis[Master], Execute := FALSE, Position := 0);
		SetStep(HomeSequence, 0);
		Home := TRUE;
END_CASE
END_METHOD

END_PROGRAM

// ---- POUs/MC3/Gearing/Support/SetStep.TcPOU
FUNCTION SetStep : UDINT
VAR_IN_OUT
	StateVar : UDINT;
END_VAR

VAR_INPUT
	NextStep : UDINT;
END_VAR

SetStep := StateVar := NextStep;

END_FUNCTION

// ---- POUs/MC3/PressToTarget/PressToTarget.TcPOU
PROGRAM PressToTarget
VAR
	bStart:				BOOL;
	
	HydAxis:			Tc3_Mc3FluidPower.AXIS_REF;
	
	fbPower:			Tc3_Mc3FluidPower.MC_Power;
	fbMoveAbsFast:		Tc3_Mc3FluidPower.MC_MoveAbsolute;
	fbMoveAbsSlow:		Tc3_Mc3FluidPower.MC_MoveAbsolute;
	fbMoveRelative:		Tc3_Mc3FluidPower.MC_MoveRelative;
	
	fbPressureCtrl:		Tc3_Mc3FluidPower.MC_LoadControl;

	timer:				TON;	
	
	nState: 			INT;
END_VAR


fbPower
(
	Axis:=HydAxis,
	Enable:=TRUE,
	EnableNegative:=TRUE,
	EnablePositive:=TRUE
);
CASE nState OF
	0:
	IF 	bStart THEN
		fbMoveAbsFast.Position:=200.0;
		fbMoveAbsFast.Velocity:=80.0;
		fbMoveAbsFast.BufferMode:=Tc3_Mc3Ptp.EBufferMode.Aborting;
		fbMoveAbsFast.Execute:=TRUE;

		fbMoveAbsSlow.Position:=201.0;
		fbMoveAbsSlow.Velocity:=2.0;
		fbMoveAbsSlow.BufferMode:=Tc3_Mc3Ptp.EBufferMode.Buffered;
		fbMoveAbsSlow.Execute:=TRUE;
		
		nState:=1;
		bStart:=false;
	END_IF
	
	1:
	nState:=2;

	2:
	IF HydAxis.McToPlc.Set.Position > fbMoveAbsFast.Position THEN
		fbPressureCtrl.Load:=300.0;
		fbPressureCtrl.Execute:=TRUE;

		nState:=3;
	END_IF
	
	3:
	fbPressureCtrl.Execute:=FALSE;
	fbMoveAbsSlow.Execute:=FALSE;
	fbMoveAbsFast.Execute:=FALSE;
	IF 	fbPressureCtrl.InLoad THEN
		timer.PT:=T#1S;
		timer.IN:=TRUE;
		nState:=4;
	END_IF
	
	4:
	IF timer.Q THEN
		fbPressureCtrl.Load:=0.0;
		fbPressureCtrl.Execute:=TRUE;
		nState:=5;
	END_IF


	5:
	IF 	fbPressureCtrl.InLoad THEN
// 		fbMoveRelative.Distance:=-5;
// 		fbMoveRelative.Velocity:=5.0;
// 		fbMoveRelative.Execute:=TRUE;
//		fbMoveAbsSlow.Position:=195;
		fbMoveAbsSlow.Position:=180;
		fbMoveAbsSlow.Velocity:=5.0;
		fbMoveAbsSlow.BufferMode:=Tc3_Mc3Ptp.EBufferMode.Aborting;
		fbMoveAbsSlow.Execute:=TRUE;

// 		fbMoveAbsFast.Position:=0.0;
// 		fbMoveAbsFast.Velocity:=50.0;
// 		fbMoveAbsFast.BufferMode:=Tc3_Mc3Ptp.EBufferMode.BlendingLow;
// 		fbMoveAbsFast.Execute:=TRUE;

		nState:=6;
	END_IF
	
	6:
	IF HydAxis.McToPlc.Set.Position < 198 THEN
		fbMoveAbsFast.Position:=0.0;
		fbMoveAbsFast.Velocity:=50.0;
		fbMoveAbsFast.BufferMode:=Tc3_Mc3Ptp.EBufferMode.Aborting;
		fbMoveAbsFast.Execute:=TRUE;
		nState:=7;
	end_if

	7:
	IF fbMoveAbsFast.Done THEN
		timer.IN:=FALSE;
		fbPressureCtrl.Execute:=FALSE;
		fbMoveAbsSlow.Execute:=FALSE;
		fbMoveAbsFast.Execute:=FALSE;
		nState:=0;
	END_IF	
END_CASE



timer();

fbMoveAbsFast
(
	Axis:=HydAxis,
);

fbMoveAbsSlow
(
	Axis:=HydAxis,
);

fbMoveRelative
(
	Axis:=HydAxis,
);


fbPressureCtrl
(
	Axis:=HydAxis,
	LoadRamp:=8000.0,
	LoadRampDerivative:=100000.0
);

END_PROGRAM

// ---- POUs/MC3/LoadControl/LoadControl.TcPOU
PROGRAM LoadControl
VAR
	bStart:				BOOL;
	
	HydAxis:			Tc3_Mc3FluidPower.AXIS_REF;
	
	fbPower:			Tc3_Mc3FluidPower.MC_Power;
	fbMoveAbsFast:		Tc3_Mc3FluidPower.MC_MoveAbsolute;
	fbMoveAbsSlow:		Tc3_Mc3FluidPower.MC_MoveAbsolute;
	
	fbPressureCtrl:		Tc3_Mc3FluidPower.MC_LoadControl;
	
	timer:				TON;	
	
	nState: 			INT;
END_VAR

fbPower
(
	Axis:=HydAxis,
	Enable:=TRUE,
	EnableNegative:=TRUE,
	EnablePositive:=TRUE
);
CASE nState OF
	0:
	IF 	bStart THEN
		fbMoveAbsFast.Position:=100.0;
		fbMoveAbsFast.Velocity:=80.0;
		fbMoveAbsFast.BufferMode:=Tc3_Mc3Ptp.EBufferMode.Aborting;
		fbMoveAbsFast.Execute:=TRUE;

		fbMoveAbsSlow.Position:=200.0;
		fbMoveAbsSlow.Velocity:=2.0;
		fbMoveAbsSlow.BufferMode:=Tc3_Mc3Ptp.EBufferMode.Buffered;
		fbMoveAbsSlow.Execute:=TRUE;

		nState:=1;
		bStart:=false;
	END_IF
	
	1:
	nState:=2;

	2:
	IF HydAxis.McToPlc.LoadControl.Act.Value > 10.0 THEN
		fbPressureCtrl.Load:=100.0;
		fbPressureCtrl.Execute:=TRUE;

		nState:=3;
	END_IF
	
	3:
	fbPressureCtrl.Execute:=FALSE;
	fbMoveAbsSlow.Execute:=FALSE;
	fbMoveAbsFast.Execute:=FALSE;
	IF 	fbPressureCtrl.InLoad THEN
		timer.PT:=T#1S;
		timer.IN:=TRUE;
		nState:=4;
	ELSIF HydAxis.McToPlc.Set.Position > 140.0 THEN
		fbMoveAbsFast.Position:=0.0;
		fbMoveAbsFast.Velocity:=50.0;
		fbMoveAbsFast.BufferMode:=Tc3_Mc3Ptp.EBufferMode.Aborting;

		fbMoveAbsFast.Execute:=TRUE;
		nState:=6;
	END_IF
	
	4:
	IF timer.Q THEN
		fbPressureCtrl.Load:=10.0;
		fbPressureCtrl.Execute:=TRUE;
		nState:=5;
	END_IF


	5:
	IF 	fbPressureCtrl.InLoad THEN
		fbMoveAbsFast.Position:=0.0;
		fbMoveAbsFast.Velocity:=50.0;

		fbMoveAbsFast.Execute:=TRUE;
		nState:=6;
	END_IF
	
	6:
	nState:=7;

	7:
	IF fbMoveAbsFast.Done THEN
		timer.IN:=FALSE;
		fbPressureCtrl.Execute:=FALSE;
		fbMoveAbsSlow.Execute:=FALSE;
		fbMoveAbsFast.Execute:=FALSE;
		nState:=0;
	END_IF	
END_CASE



timer();

fbMoveAbsFast
(
	Axis:=HydAxis,
);

fbMoveAbsSlow
(
	Axis:=HydAxis,
);


fbPressureCtrl
(
	Axis:=HydAxis,
	LoadRamp:=50.0,
	LoadRampDerivative:=50.0
);

END_PROGRAM

// ---- POUs/MC3/Gearing/Support/CompareLREAL.TcPOU
FUNCTION CompareLREAL : BOOL
VAR_INPUT
	Var1	: LREAL;
	Var2	: LREAL;
	Epsilon : LREAL := 1E-6;
END_VAR

CompareLREAL := ABS(Var1 - Var2) < Epsilon;

END_FUNCTION
